Universal Robots PolyScope program: 04_Pick_Place_04_Loop_if.urp

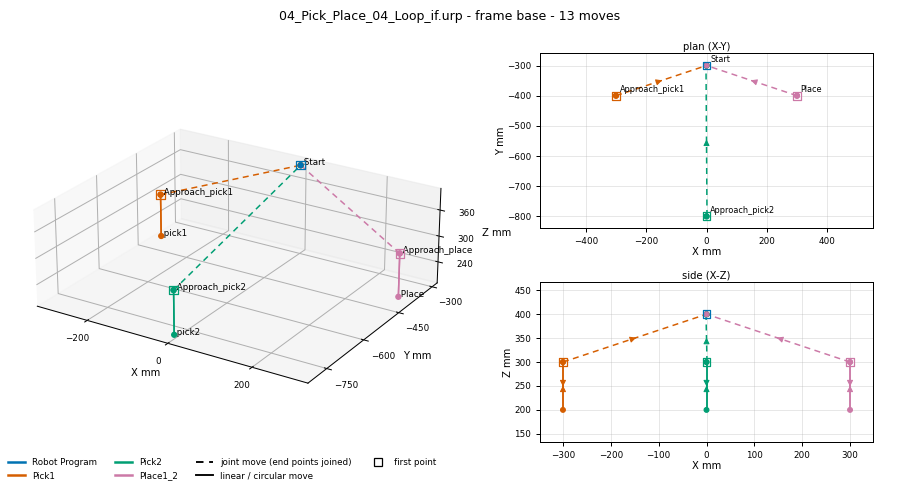
[picture p0: tool path of 04_Pick_Place_04_Loop_if.urp in frame base, 13 of 13 moves have a stored position in this frame; points joined in program order, loops and branches not executed]
Program 04_Pick_Place_04_Loop_if (installation=default directory=/home/ur/ursim-current/programs/Test_Programs createdIn=5.9.1.1031110 lastSavedIn=5.9.1.1031110 robotSerialNumber=20195599999)
Calibrated DH parameters: a=[0, -0.425, -0.3922, 0, 0, 0]; d=[0.1625, 0, 0, 0.1333, 0.0997, 0.0996]; alpha=[1.570796, 0, 0, 1.570796, -1.570796, 0]; deltaTheta=[0, 0, 0, 0, 0, 0]
Robot Program (runOnlyOnce=false)
  'Init program'
  MoveJ speed 60 deg/s, acceleration 80 deg/s^2 (useActiveTCP=true) feature=Base
    Waypoint Start: TCP in base x=0 y=-300 z=400 mm, rx=0 ry=3.1416 rz=0 rad; joints [-63.619, -58.456, -125.213, -86.33, 90, 26.381] deg
  Loop Counting (count=3) loopVariable(name=Loop_1)
    If digital_in[0]≟ True
      Call Pick1
    Else 
      Call Pick2
    Call Place1_2
    Call LED
SubProgram -> Pick1
SubProgram -> Pick2
SubProgram -> Place1_2
SubProgram -> LED
SubProgram Pick1 (keepSynchronizedWithDisk=false)
  Folder Pick1
    MoveJ speed 60 deg/s, acceleration 80 deg/s^2 (useActiveTCP=true) feature=Base
      Waypoint Approach_pick1: TCP in base x=-300 y=-400 z=300 mm, rx=0 ry=3.1416 rz=0 rad; joints [-111.408, -95.003, -113.354, -61.643, 90, -21.408] deg; TCP offset x=0 y=0 z=0 mm, rx=0 ry=0 rz=0 rad
    MoveL speed 250 mm/s, acceleration 1200 mm/s^2 (useActiveTCP=true) feature=Base
      Waypoint pick1: TCP in base x=-300 y=-400 z=200 mm, rx=0 ry=3.1416 rz=0 rad; joints [-111.408, -104.003, -120.574, -45.423, 90, -21.408] deg
      Set SingleDigitalPulseActionState SingleDigitalPulseActionState(hiPulseInSeconds=0.5, pin=digital_out[0])
      Waypoint Approach_pick1: TCP in base x=-300 y=-400 z=300 mm, rx=0 ry=3.1416 rz=0 rad; joints [-111.408, -95.003, -113.354, -61.643, 90, -21.408] deg; TCP offset x=0 y=0 z=0 mm, rx=0 ry=0 rz=0 rad
    MoveJ speed 60 deg/s, acceleration 80 deg/s^2 (useActiveTCP=true) feature=Base
      Waypoint Start: TCP in base x=0 y=-300 z=400 mm, rx=0 ry=3.1416 rz=0 rad; joints [-63.619, -58.456, -125.213, -86.33, 90, 26.381] deg
SubProgram Pick2 (keepSynchronizedWithDisk=false)
  Folder Pick2
    MoveJ speed 60 deg/s, acceleration 80 deg/s^2 (useActiveTCP=true) feature=Base
      Waypoint Approach_pick2: TCP in base x=0 y=-800 z=300 mm, rx=0 ry=3.1416 rz=0 rad; joints [-80.408, -135.256, -53.851, -80.893, 90, 9.592] deg; TCP offset x=0 y=0 z=0 mm, rx=0 ry=0 rz=0 rad
    MoveL speed 250 mm/s, acceleration 1200 mm/s^2 (useActiveTCP=true) feature=Base
      Waypoint pick2: TCP in base x=0 y=-800 z=200 mm, rx=0 ry=3.1416 rz=0 rad; joints [-80.408, -139.381, -61.468, -69.151, 90, 9.592] deg; TCP offset x=0 y=0 z=0 mm, rx=0 ry=0 rz=0 rad
      Set SingleDigitalPulseActionState SingleDigitalPulseActionState(hiPulseInSeconds=0.5, pin=digital_out[0])
      Waypoint Approach_pick2: TCP in base x=0 y=-800 z=300 mm, rx=0 ry=3.1416 rz=0 rad; joints [-80.408, -135.256, -53.851, -80.893, 90, 9.592] deg; TCP offset x=0 y=0 z=0 mm, rx=0 ry=0 rz=0 rad
    MoveJ speed 60 deg/s, acceleration 80 deg/s^2 (useActiveTCP=true) feature=Base
      Waypoint Start: TCP in base x=0 y=-300 z=400 mm, rx=0 ry=3.1416 rz=0 rad; joints [-63.619, -58.456, -125.213, -86.33, 90, 26.381] deg
SubProgram Place1_2 (keepSynchronizedWithDisk=false)
  Folder Place
    MoveJ speed 60 deg/s, acceleration 80 deg/s^2 (useActiveTCP=true) feature=Base
      Waypoint Approach_place: TCP in base x=300 y=-400 z=300 mm, rx=0 ry=3.1416 rz=0 rad; joints [-37.668, -95.003, -113.354, -61.643, 90, 52.332] deg
    MoveL speed 250 mm/s, acceleration 1200 mm/s^2 (useActiveTCP=true) feature=Base
      Waypoint Place: TCP in base x=300 y=-400 z=200 mm, rx=0 ry=3.1416 rz=0 rad; joints [-37.668, -104.003, -120.574, -45.423, 90, 52.332] deg
      Set DigitalOutput pin=digital_out[0]; digitalValue=0
      Waypoint Approach_place: TCP in base x=300 y=-400 z=300 mm, rx=0 ry=3.1416 rz=0 rad; joints [-37.668, -95.003, -113.354, -61.643, 90, 52.332] deg
    MoveJ speed 60 deg/s, acceleration 80 deg/s^2 (useActiveTCP=true) feature=Base
      Waypoint Start: TCP in base x=0 y=-300 z=400 mm, rx=0 ry=3.1416 rz=0 rad; joints [-63.619, -58.456, -125.213, -86.33, 90, 26.381] deg
SubProgram LED (keepSynchronizedWithDisk=false)
  Loop While (checkContinuously=false) expression=digital_in[1]≟ False
    Set DigitalOutput pin=digital_out[0]; digitalValue=1
    Wait Sleep waitTime=0.2
    Set DigitalOutput pin=digital_out[0]; digitalValue=0
    Wait Sleep waitTime=0.2
